// TIA Portal V16 export
// export: Created 2022-11-14T17:35:46.4739204Z, ExportSetting WithDefaults, DisplayName Totally Integrated Automation Portal, DisplayVersion V16, DisplayName TIA Portal Version Control Interface, DisplayVersion V16, DisplayName TIA Portal Openness, DisplayVersion V16, DisplayName STEP 7 Professional, DisplayVersion V16, DisplayName STEP 7 Safety, DisplayVersion V16, DisplayName WinCC Advanced, DisplayVersion V16
DATA_BLOCK "DB235_Program15"   // DB235
{ S7_Optimized_Access := 'FALSE' }
AUTHOR : Robopac
VERSION : 0.0
// stored: AutoNumber false, IsOnlyStoredInLoadMemory false, IsWriteProtectedInAS false
   VAR RETAIN
      Program15 { S7_SetPoint := 'True'} : "DatiProgramma";
   END_VAR
BEGIN
   Program15.Wrapping := TRUE;
   Program15.TopLenght := 500;
   Program15.TopRelease := 0;
   Program15.TopDown := 0;
   Program15.Top := 4;
   Program15.PressurePTime := 0;
   Program15.LifterTime := 0;
   Program15.RevOverContrast := 1;
   Program15.RopeEndCycle := 16#02;
   Program15.Spare4 := 16#01;
   Program15.RopeTime := 1500;
   Program15.RevOverClamp := 1;
   Program15.FilmForceFinalRev := 10;
   Program15.FilmPrestretchFinalRev := 100;
   Program15.ArmSpeed := 100;
   Program15.CarriageDown4Top := 500;
   Program15.TopDownTime := 1500;
   Program15.LapsUnderTop := 0;
   Program15.Spare6 := 0;
   Program15.Spare7 := 0;
   Program15.Spare8 := 0;
   Program15.Spare9 := 0;
   Program15.Spare10 := 0;
   Program15.Spare11 := 0;
   Program15.Spare12 := 0;
   Program15.Overlap0_1 := 0;
   Program15.Height1 := 130;
   Program15.Landmark1 := FALSE;
   Program15.Lifter1 := FALSE;
   Program15.SpareBit1H1 := FALSE;
   Program15.Airblower1 := TRUE;
   Program15.NextStep1 := TRUE;
   Program15.PressureP1 := TRUE;
   Program15.SpareByte2H1 := 16#00;
   Program15.Revolution1 := 1;
   Program15.RopeUnit1_1 := 16#01;
   Program15.RopeUnit1_2 := 16#01;
   Program15.FilmForce1 := 5;
   Program15.FilmPrestretch1 := 200;
   Program15.Spare3H1 := 0;
   Program15.Spare49 := 0;
   Program15.Spare50 := 0;
   Program15.Spare51 := 0;
   Program15.Spare52 := 0;
   Program15.Spare53 := 0;
   Program15.Overlap1_2 := 0;
   Program15.Height2 := 50;
   Program15.Landmark2 := FALSE;
   Program15.Lifter2 := FALSE;
   Program15.SpareBit1H2 := FALSE;
   Program15.Airblower2 := TRUE;
   Program15.NextStep2 := TRUE;
   Program15.PressureP2 := TRUE;
   Program15.SpareByte2H2 := 16#00;
   Program15.Revolution2 := 1;
   Program15.RopeUnit2_1 := 16#01;
   Program15.RopeUnit2_2 := 16#01;
   Program15.FilmForce2 := 20;
   Program15.FilmPrestretch2 := 200;
   Program15.Spare3H2 := 0;
   Program15.Spare54 := 0;
   Program15.Spare55 := 0;
   Program15.Spare56 := 0;
   Program15.Spare57 := 0;
   Program15.Spare58 := 0;
   Program15.Overlap2_3 := 100;
   Program15.Height3 := -50;
   Program15.Landmark3 := TRUE;
   Program15.Lifter3 := FALSE;
   Program15.SpareBit1H3 := FALSE;
   Program15.Airblower3 := TRUE;
   Program15.NextStep3 := TRUE;
   Program15.PressureP3 := TRUE;
   Program15.SpareByte2H3 := 16#00;
   Program15.Revolution3 := 2;
   Program15.RopeUnit3_1 := 16#01;
   Program15.RopeUnit3_2 := 16#01;
   Program15.FilmForce3 := 30;
   Program15.FilmPrestretch3 := 200;
   Program15.Spare3H3 := 0;
   Program15.Spare59 := 0;
   Program15.Spare60 := 0;
   Program15.Spare61 := 380;
   Program15.Spare62 := 2800;
   Program15.Spare63 := 0;
   Program15.Overlap3_4 := 100;
   Program15.Height4 := 100;
   Program15.Landmark4 := FALSE;
   Program15.Lifter4 := FALSE;
   Program15.SpareBit1H4 := FALSE;
   Program15.Airblower4 := TRUE;
   Program15.NextStep4 := TRUE;
   Program15.PressureP4 := TRUE;
   Program15.SpareByte2H4 := 16#00;
   Program15.Revolution4 := 3;
   Program15.RopeUnit4_1 := 16#02;
   Program15.RopeUnit4_2 := 16#02;
   Program15.FilmForce4 := 30;
   Program15.FilmPrestretch4 := 200;
   Program15.Spare3H4 := 0;
   Program15.Spare64 := 0;
   Program15.Spare65 := 0;
   Program15.Spare66 := 0;
   Program15.Spare67 := 0;
   Program15.Spare68 := 0;
   Program15.Overlap4_5 := 0;
   Program15.Height5 := 50;
   Program15.Landmark5 := FALSE;
   Program15.Lifter5 := FALSE;
   Program15.SpareBit1H5 := FALSE;
   Program15.Airblower5 := TRUE;
   Program15.NextStep5 := FALSE;
   Program15.PressureP5 := FALSE;
   Program15.SpareByte2H5 := 16#00;
   Program15.Revolution5 := 1;
   Program15.RopeUnit5_1 := 16#01;
   Program15.RopeUnit5_2 := 16#01;
   Program15.FilmForce5 := 30;
   Program15.FilmPrestretch5 := 200;
   Program15.Spare3H5 := 0;
   Program15.Spare69 := 0;
   Program15.Spare70 := 0;
   Program15.Spare71 := 0;
   Program15.Spare72 := 0;
   Program15.Spare73 := 0;
   Program15.Overlap5_6 := 100;
   Program15.Height6 := 50;
   Program15.Landmark6 := FALSE;
   Program15.Lifter6 := FALSE;
   Program15.SpareBit1H6 := FALSE;
   Program15.Airblower6 := TRUE;
   Program15.NextStep6 := FALSE;
   Program15.PressureP6 := FALSE;
   Program15.SpareByte2H6 := 16#00;
   Program15.Revolution6 := 2;
   Program15.RopeUnit6_1 := 16#02;
   Program15.RopeUnit6_2 := 16#01;
   Program15.FilmForce6 := 20;
   Program15.FilmPrestretch6 := 200;
   Program15.Spare3H6 := 0;
   Program15.Spare74 := 0;
   Program15.Spare75 := 0;
   Program15.Spare76 := 0;
   Program15.Spare77 := 0;
   Program15.Spare78 := 0;
   Program15.Overlap6_7 := 0;
   Program15.Height7 := 0;
   Program15.Landmark7 := FALSE;
   Program15.Lifter7 := FALSE;
   Program15.SpareBit1H7 := FALSE;
   Program15.Airblower7 := FALSE;
   Program15.NextStep7 := TRUE;
   Program15.PressureP7 := FALSE;
   Program15.SpareByte2H7 := 16#00;
   Program15.Revolution7 := 1;
   Program15.RopeUnit7_1 := 16#01;
   Program15.RopeUnit7_2 := 16#01;
   Program15.FilmForce7 := 0;
   Program15.FilmPrestretch7 := 100;
   Program15.Spare3H7 := 0;
   Program15.Spare79 := 0;
   Program15.Spare80 := 0;
   Program15.Spare81 := 0;
   Program15.Spare82 := 0;
   Program15.Spare83 := 0;
   Program15.Overlap7_8 := 0;
   Program15.Height8 := 0;
   Program15.Landmark8 := FALSE;
   Program15.Lifter8 := FALSE;
   Program15.SpareBit1H8 := FALSE;
   Program15.Airblower8 := FALSE;
   Program15.NextStep8 := TRUE;
   Program15.PressureP8 := FALSE;
   Program15.SpareByte2H8 := 16#00;
   Program15.Revolution8 := 1;
   Program15.RopeUnit8_1 := 16#01;
   Program15.RopeUnit8_2 := 16#01;
   Program15.FilmForce8 := 0;
   Program15.FilmPrestretch8 := 100;
   Program15.Spare3H8 := 0;
   Program15.Spare84 := 0;
   Program15.Spare85 := 0;
   Program15.Spare86 := 0;
   Program15.Spare87 := 0;
   Program15.Spare88 := 0;
   Program15.Overlap8_9 := 0;
   Program15.Height9 := 0;
   Program15.Landmark9 := FALSE;
   Program15.Lifter9 := FALSE;
   Program15.SpareBit1H9 := FALSE;
   Program15.Airblower9 := FALSE;
   Program15.NextStep9 := TRUE;
   Program15.PressureP9 := FALSE;
   Program15.SpareByte2H9 := 16#00;
   Program15.Revolution9 := 1;
   Program15.RopeUnit9_1 := 16#01;
   Program15.RopeUnit9_2 := 16#01;
   Program15.FilmForce9 := 0;
   Program15.FilmPrestretch9 := 100;
   Program15.Spare3H9 := 0;
   Program15.Spare89 := 0;
   Program15.Spare90 := 0;
   Program15.Spare91 := 0;
   Program15.Spare92 := 0;
   Program15.Spare93 := 0;
   Program15.Overlap9_10 := 0;
   Program15.Height10 := 0;
   Program15.Landmark10 := FALSE;
   Program15.Lifter10 := FALSE;
   Program15.SpareBit1H10 := FALSE;
   Program15.Airblower10 := FALSE;
   Program15.NextStep10 := FALSE;
   Program15.PressureP10 := FALSE;
   Program15.SpareByte2H10 := 16#00;
   Program15.Revolution10 := 1;
   Program15.RopeUnit10_1 := 16#01;
   Program15.RopeUnit10_2 := 16#01;
   Program15.FilmForce10 := 0;
   Program15.FilmPrestretch10 := 100;
   Program15.Spare3H10 := 0;
   Program15.Spare94 := 0;
   Program15.Spare95 := 0;
   Program15.Spare96 := 0;
   Program15.Spare97 := 0;
   Program15.Spare98 := 0;
   Program15.Overlap10_11 := 0;
   Program15.Height11 := 0;
   Program15.Landmark11 := FALSE;
   Program15.Lifter11 := FALSE;
   Program15.SpareBit1H11 := FALSE;
   Program15.Airblower11 := FALSE;
   Program15.NextStep11 := TRUE;
   Program15.PressureP11 := FALSE;
   Program15.SpareByte2H11 := 16#00;
   Program15.Revolution11 := 1;
   Program15.RopeUnit11_1 := 16#01;
   Program15.RopeUnit11_2 := 16#01;
   Program15.FilmForce11 := 0;
   Program15.FilmPrestretch11 := 100;
   Program15.Spare3H11 := 0;
   Program15.Spare99 := 0;
   Program15.Spare100 := 0;
   Program15.Spare101 := 0;
   Program15.Spare102 := 0;
   Program15.Spare103 := 0;
   Program15.Overlap11_12 := 0;
   Program15.Height12 := 0;
   Program15.Landmark12 := FALSE;
   Program15.Lifter12 := FALSE;
   Program15.SpareBit1H12 := FALSE;
   Program15.Airblower12 := FALSE;
   Program15.NextStep12 := FALSE;
   Program15.PressureP12 := FALSE;
   Program15.SpareByte2H12 := 16#00;
   Program15.Revolution12 := 1;
   Program15.RopeUnit12_1 := 16#01;
   Program15.RopeUnit12_2 := 16#01;
   Program15.FilmForce12 := 0;
   Program15.FilmPrestretch12 := 100;
   Program15.Spare3H12 := 0;
   Program15.Spare104 := 0;
   Program15.Spare105 := 0;
   Program15.Spare106 := 0;
   Program15.Spare107 := 0;
   Program15.Spare108 := 0;
END_DATA_BLOCK
